{attribute addProperty BoxType "EL6695-0000-0001"}
{attribute addProperty Id "TxPDO_toggleAT %I*BOOL811TxPDO_stateAT %I*BOOL812External_device_not_connectedAT %I*BOOL8116"}
{attribute addProperty CRC "3091651366"}
{attribute addProperty SizeInBites "24"}
{attribute addProperty SizeInBytes "3"}
TYPE SYNC_Inputs_B846DB26 :
STRUCT
	{attribute addProperty Name "TxPDO_toggle"}
	TxPDO_toggle AT %I* : BOOL;
	{attribute addProperty Name "TxPDO_state"}
	TxPDO_state AT %I* : BOOL;
	{attribute addProperty Name "External_device_not_connected"}
	External_device_not_connected AT %I* : BOOL;
END_STRUCT
END_TYPE

(* stored: Version 1.2.0.0, ProductVersion 3.1.4024.9
   DUT SYNC_Inputs_B846DB26: Id {d75fbadc-c1f0-41a5-8088-ce2775228330} *)
